(*
SPDX-FileCopyrightText: © 2026 Oleksandr Tiutyk <trofimich@gmail.com>
SPDX-License-Identifier: MIT
License: https://opensource.org/license/mit
*)

(*!
<summary>Converts angular values between degrees and radians.</summary>
<description>
Uses LREAL arithmetic and the PI constant from Tc2_System. Conversion does not normalize angles to a single
revolution or perform argument validation.
</description>
*)

PROGRAM Trigonometry
VAR
	{attribute 'hide'} 
	_ClassName : STRING := __POUNAME();
END_VAR

{attribute 'monitoring' := 'call'}
PROPERTY ClassName : REFERENCE TO STRING
GET
ClassName REF= _ClassName;
END_GET
END_PROPERTY

(*!
<summary>Converts an angle in degrees to radians.</summary>
<description>
Multiplies by PI and divides by 180 using LREAL arithmetic, including its precision and range limits.
</description>
<param name="degrees">Angle expressed in degrees.</param>
*)
METHOD ConvertDegreesToRadians : LREAL
VAR_INPUT
	degrees : LREAL;
END_VAR
ConvertDegreesToRadians := degrees * Tc2_System.Global_Variables.PI / 180;
END_METHOD

(*!
<summary>Converts an angle in radians to degrees.</summary>
<description>
Multiplies by 180 and divides by PI using LREAL arithmetic, including its precision and range limits.
</description>
<param name="radians">Angle expressed in radians.</param>
*)
METHOD ConvertRadiansToDegrees : LREAL
VAR_INPUT
	radians : LREAL;
END_VAR
ConvertRadiansToDegrees := radians * 180 / Tc2_System.Global_Variables.PI;
END_METHOD

(*!
<summary>Provides the library namespace used in diagnostics.</summary>
<description>
Borrowed read-only reference to the compiler-initialized library namespace; no ownership transfer.
</description>
*)
{attribute 'monitoring' := 'call'}
PROPERTY NamespaceName : REFERENCE TO STRING
GET
NamespaceName REF= CurrentNamespace.Name;
END_GET
END_PROPERTY

END_PROGRAM

(* stored: Version 1.1.0.1
   POU Trigonometry: Id {2c342da1-0c2d-4d9a-b590-c322f1e48840}, SpecialFunc None
   Property ClassName: Id {4066085f-a03d-4767-943f-a4a2ac75f162}
   Get Get: Id {5348d100-2fe7-4170-ba36-e606066e8cce}
   Method ConvertDegreesToRadians: Id {00966382-7173-42f2-a216-84e52e8a6a77}
   Method ConvertRadiansToDegrees: Id {28142a7d-b968-41ed-84a3-710729c3981e}
   Property NamespaceName: Id {a3e5efee-a8fa-4c2d-8dfc-5d099e702df3}
   Get Get: Id {c0487467-7977-4fdc-9e7b-2b228a7ef86a} *)
